PROGRAM MAIN_Shutdown
VAR
END_VAR

Shutdown();

END_PROGRAM

(* stored: Version 1.1.0.1, ProductVersion 3.1.4022.3
   POU MAIN_Shutdown: Id {0b3b2413-2c53-4ea2-9d0c-46842e409463}, SpecialFunc None *)
